TYPE DigitalInputBase_50022E7B :
STRUCT
END_STRUCT
END_TYPE

(* stored: Version 1.2.0.0, ProductVersion 3.1.4024.9
   DUT DigitalInputBase_50022E7B: Id {490ce627-f6b0-4dbe-b056-52c7bb47fb49} *)
